// TIA Portal V17 export
// export: Created 2022-07-28T18:02:47.9991032Z, ExportSetting None, DisplayName Totally Integrated Automation Portal, DisplayVersion V17, DisplayName TIA Portal Openness, DisplayVersion V17, DisplayName TIA Portal Teamcenter Gateway, DisplayVersion V17, DisplayName TIA Portal Version Control Interface, DisplayVersion V17, DisplayName TIA Portal Test Suite Advanced, DisplayVersion V17, DisplayName SINAMICS Startdrive Advanced, DisplayVersion V17, DisplayName SINAMICS DCC, DisplayVersion V17, DisplayName SINAMICS Startdrive G130, G150, S120, S150, SINAMICS MV, S210, DisplayVersion V17, DisplayName SINAMICS Startdrive G110M, G120, G120C, G120D, G120P, G115D, DisplayVersion V17, DisplayName STEP 7 Professional, DisplayVersion V17, DisplayName SIMATIC Energy Suite, DisplayVersion V17, DisplayName STEP 7 CFC, DisplayVersion V17, DisplayName STEP 7 Safety, DisplayVersion V17, DisplayName WinCC Advanced / Unified PC, DisplayVersion V17, DisplayName SIMATIC Visualization Architect, DisplayVersion V17
FUNCTION "Field_FC" : Void   // FC19, SCL
{ S7_Optimized_Access := 'TRUE' }
// stored: SetENOAutomatically false
   VAR_TEMP
      t_SupplyRelease : Bool;   // 1 - Release from supply
   END_VAR
BEGIN
   #t_SupplyRelease := true;

   REGION (ID = 1) Витратомір пари на нову рафінацію Steam Flowmeter New
       //Тип елемента: Аналоговий витратомір
       //Параметри давача: Scale=; 4-20mA; Analog = 0 - 27648;
       //Одиниці вимірювання: m3/h
       //Додаткова інформація: SITRANS FX330 / 7ME2610-3LD00-0AA0-Z

       REGION Блок керування       
           "D_SteamFlowmeterNew_FT1_Ctrl"(I_Initialization := "D_General_ProgramDATA".RestartPLC,
                                          IR_Raw := "D_InOut"."SteamFlowmeterNew_FT1".II_AnalogValue,
                                          IR_Coef:=60.0,
                                          II_Mode := 0,
                                          I_GlobalRST := "D_General_ProgramDATA".ResetGlobal,
                                          I_Puls_1s:="D_PLC".PLS.P1S,
                                          IR_CycleTime := "D_PLC".TIME_TCK.cyclic_sec_R,
                                          II_Obj_ID := 1,
                                          IQ_PLC_CycleInfo := "D_PLC_CycleInfo_DATA".Grp_Obj[1, 0]);
       END_REGION

   END_REGION

   REGION (ID = 2) Витратомір пари на стару рафінацію Steam Flowmeter Old
       //Тип елемента: Аналоговий витратомір
       //Параметри давача: Scale=; 4-20mA; Analog = 0 - 27648;
       //Одиниці вимірювання: m3/h
       //Додаткова інформація: SITRANS FX330 / 7ME2610-3LD00-0AA0-Z

       REGION Блок керування       
           "D_SteamFlowmeterOld_FT1_Ctrl"(I_Initialization := "D_General_ProgramDATA".RestartPLC,
                                          IR_Raw := "D_InOut"."SteamFlowmeterOld_FT1".II_AnalogValue,
                                          IR_Coef:=60.0,
                                          II_Mode := 0,
                                          I_GlobalRST := "D_General_ProgramDATA".ResetGlobal,
                                          I_Puls_1s:="D_PLC".PLS.P1S,
                                          IR_CycleTime := "D_PLC".TIME_TCK.cyclic_sec_R,
                                          II_Obj_ID := 2,
                                          IQ_PLC_CycleInfo := "D_PLC_CycleInfo_DATA".Grp_Obj[1, 0]);
       END_REGION

   END_REGION

   REGION (ID = 3) Перетворювач тиску обор.води PTНГр
       //Тип елемента: Аналоговий сигнал
       //Параметри давача: Scale=0-10bar; 4-20mA; Analog = 0 - 27648;
       //Одиниці вимірювання: bar
       //Додаткова інформація: 

       REGION Блок керування       
           "D_PTNGr_PT1_Ctrl"(I_Initialization := "D_General_ProgramDATA".RestartPLC,
                              IR_Raw := "D_InOut"."PTNGr_PT1".II_AnalogValue,
                              II_Mode := 0,
                              I_GlobalRST := "D_General_ProgramDATA".ResetGlobal,
                              IR_CycleTime := "D_PLC".TIME_TCK.cyclic_sec_R,
                              II_Obj_ID := 3,
                              IQ_PLC_CycleInfo := "D_PLC_CycleInfo_DATA".Grp_Obj[1, 0]);
       END_REGION

   END_REGION

   REGION (ID = 4) Перетворювач температури вих.води ХМ1 ТТW1011
       //Тип елемента: Аналоговий сигнал
       //Параметри давача: Scale=0-150C; 4-20mA; Analog = 0 - 27648;
       //Одиниці вимірювання: C
       //Додаткова інформація: 

       REGION Блок керування       
           "D_TTW1011_TT1_Ctrl"(I_Initialization := "D_General_ProgramDATA".RestartPLC,
                                IR_Raw := "D_InOut"."TTW1011_TT1".II_AnalogValue,
                                II_Mode := 0,
                                I_GlobalRST := "D_General_ProgramDATA".ResetGlobal,
                                IR_CycleTime := "D_PLC".TIME_TCK.cyclic_sec_R,
                                II_Obj_ID := 4,
                                IQ_PLC_CycleInfo := "D_PLC_CycleInfo_DATA".Grp_Obj[1, 0]);
       END_REGION

   END_REGION

   REGION (ID = 5) Перетворювач температури вих.води ХМ2 TT811
       //Тип елемента: Аналоговий сигнал
       //Параметри давача: Scale=0-150C; 4-20mA; Analog = 0 - 27648;
       //Одиниці вимірювання: C
       //Додаткова інформація: 

       REGION Блок керування       
           "D_TT811_TT1_Ctrl"(I_Initialization := "D_General_ProgramDATA".RestartPLC,
                              IR_Raw := "D_InOut"."TT811_TT1".II_AnalogValue,
                              II_Mode := 0,
                              I_GlobalRST := "D_General_ProgramDATA".ResetGlobal,
                              IR_CycleTime := "D_PLC".TIME_TCK.cyclic_sec_R,
                              II_Obj_ID := 5,
                              IQ_PLC_CycleInfo := "D_PLC_CycleInfo_DATA".Grp_Obj[1, 0]);
       END_REGION

   END_REGION

   REGION (ID = 6) Перетворювач тиску (рівень басейну градирні 1) LTБ1Гр
       //Тип елемента: Аналоговий сигнал
       //Параметри давача: Scale=0-0.25bar; 4-20mA; Analog = 0 - 27648;
       //Одиниці вимірювання: м
       //Додаткова інформація: 

       REGION Блок керування       
           "D_LTB1Gr_LT1_Ctrl"(I_Initialization := "D_General_ProgramDATA".RestartPLC,
                               IR_Raw := "D_InOut"."LTB1Gr_LT1".II_AnalogValue,
                               II_Mode := 0,
                               I_GlobalRST := "D_General_ProgramDATA".ResetGlobal,
                               IR_CycleTime := "D_PLC".TIME_TCK.cyclic_sec_R,
                               II_Obj_ID := 6,
                               IQ_PLC_CycleInfo := "D_PLC_CycleInfo_DATA".Grp_Obj[1, 0]);
       END_REGION

   END_REGION

   REGION (ID = 7) Перетворювач тиску (рівень басейну градирні 2) LTБ2Гр
       //Тип елемента: Аналоговий сигнал
       //Параметри давача: Scale=0-0.25bar; 4-20mA; Analog = 0 - 27648;
       //Одиниці вимірювання: м
       //Додаткова інформація: 
       //"D_LTB1Gr_LT1_HMI".Config.r_Offset := 1.0;
       REGION Блок керування       
           "D_LTB2Gr_LT1_Ctrl"(I_Initialization := "D_General_ProgramDATA".RestartPLC,
                               IR_Raw := "D_InOut"."LTB2Gr_LT1".II_AnalogValue,
                               II_Mode := 0,
                               I_GlobalRST := "D_General_ProgramDATA".ResetGlobal,
                               IR_CycleTime := "D_PLC".TIME_TCK.cyclic_sec_R,
                               II_Obj_ID := 7,
                               IQ_PLC_CycleInfo := "D_PLC_CycleInfo_DATA".Grp_Obj[1, 0]);
       END_REGION

   END_REGION

   REGION (ID = 8) Аналоговий сигнал від AirForce 1 G1
       //Тип елемента: Аналоговий сигнал
       //Параметри давача: Scale= ; 4-20mA; Analog = 0 - 27648;
       //Одиниці вимірювання: 
       //Додаткова інформація: 

       REGION Блок керування       
           "D_G1_AI1_Ctrl"(I_Initialization := "D_General_ProgramDATA".RestartPLC,
                           IR_Raw := "D_InOut"."G1_AI1".II_AnalogValue,
                           II_Mode := 0,
                           I_GlobalRST := "D_General_ProgramDATA".ResetGlobal,
                           IR_CycleTime := "D_PLC".TIME_TCK.cyclic_sec_R,
                           II_Obj_ID := 8,
                           IQ_PLC_CycleInfo := "D_PLC_CycleInfo_DATA".Grp_Obj[1, 0]);
       END_REGION

   END_REGION

   REGION (ID = 9) Аналоговий сигнал від AirForce 2 G1
       //Тип елемента: Аналоговий сигнал
       //Параметри давача: Scale= ; 4-20mA; Analog = 0 - 27648;
       //Одиниці вимірювання: 
       //Додаткова інформація: 

       REGION Блок керування       
           "D_G1_AI2_Ctrl"(I_Initialization := "D_General_ProgramDATA".RestartPLC,
                           IR_Raw := "D_InOut"."G1_AI2".II_AnalogValue,
                           II_Mode := 0,
                           I_GlobalRST := "D_General_ProgramDATA".ResetGlobal,
                           IR_CycleTime := "D_PLC".TIME_TCK.cyclic_sec_R,
                           II_Obj_ID := 9,
                           IQ_PLC_CycleInfo := "D_PLC_CycleInfo_DATA".Grp_Obj[1, 0]);
       END_REGION

   END_REGION

   REGION (ID = 10) Аналоговий сигнал від AirForce 3 G1
       //Тип елемента: Аналоговий сигнал
       //Параметри давача: Scale= ; 4-20mA; Analog = 0 - 27648;
       //Одиниці вимірювання: 
       //Додаткова інформація: 

       REGION Блок керування       
           "D_G1_AI3_Ctrl"(I_Initialization := "D_General_ProgramDATA".RestartPLC,
                           IR_Raw := "D_InOut"."G1_AI3".II_AnalogValue,
                           II_Mode := 0,
                           I_GlobalRST := "D_General_ProgramDATA".ResetGlobal,
                           IR_CycleTime := "D_PLC".TIME_TCK.cyclic_sec_R,
                           II_Obj_ID := 10,
                           IQ_PLC_CycleInfo := "D_PLC_CycleInfo_DATA".Grp_Obj[1, 0]);
       END_REGION

   END_REGION

   REGION (ID = 11) Аналоговий сигнал від AirForce 4 G1
       //Тип елемента: Аналоговий сигнал
       //Параметри давача: Scale= ; 4-20mA; Analog = 0 - 27648;
       //Одиниці вимірювання: 
       //Додаткова інформація: 

       REGION Блок керування       
           "D_G1_AI4_Ctrl"(I_Initialization := "D_General_ProgramDATA".RestartPLC,
                           IR_Raw := "D_InOut"."G1_AI4".II_AnalogValue,
                           II_Mode := 0,
                           I_GlobalRST := "D_General_ProgramDATA".ResetGlobal,
                           IR_CycleTime := "D_PLC".TIME_TCK.cyclic_sec_R,
                           II_Obj_ID := 11,
                           IQ_PLC_CycleInfo := "D_PLC_CycleInfo_DATA".Grp_Obj[1, 0]);
       END_REGION

   END_REGION

   REGION (ID = 12) Аналоговий сигнал від AirForce 5 G1
       //Тип елемента: Аналоговий сигнал
       //Параметри давача: Scale= ; 4-20mA; Analog = 0 - 27648;
       //Одиниці вимірювання: 
       //Додаткова інформація: 

       REGION Блок керування       
           "D_G1_AI5_Ctrl"(I_Initialization := "D_General_ProgramDATA".RestartPLC,
                           IR_Raw := "D_InOut"."G1_AI5".II_AnalogValue,
                           II_Mode := 0,
                           I_GlobalRST := "D_General_ProgramDATA".ResetGlobal,
                           IR_CycleTime := "D_PLC".TIME_TCK.cyclic_sec_R,
                           II_Obj_ID := 12,
                           IQ_PLC_CycleInfo := "D_PLC_CycleInfo_DATA".Grp_Obj[1, 0]);
       END_REGION

   END_REGION

   REGION (ID = 13) Аналоговий сигнал від AirForce 6 G1
       //Тип елемента: Аналоговий сигнал
       //Параметри давача: Scale= ; 4-20mA; Analog = 0 - 27648;
       //Одиниці вимірювання: 
       //Додаткова інформація: 

       REGION Блок керування       
           "D_G1_AI6_Ctrl"(I_Initialization := "D_General_ProgramDATA".RestartPLC,
                           IR_Raw := "D_InOut"."G1_AI6".II_AnalogValue,
                           II_Mode := 0,
                           I_GlobalRST := "D_General_ProgramDATA".ResetGlobal,
                           IR_CycleTime := "D_PLC".TIME_TCK.cyclic_sec_R,
                           II_Obj_ID := 13,
                           IQ_PLC_CycleInfo := "D_PLC_CycleInfo_DATA".Grp_Obj[1, 0]);
       END_REGION

   END_REGION

   REGION (ID = 14) Перетворювач тиску (рівень ємності конденсату) LT R46
       //Тип елемента: Аналоговий сигнал
       //Параметри давача: Scale=0-0.4bar; 4-20mA; Analog = 0 - 27648;
       //Одиниці вимірювання: м
       //Додаткова інформація: 

       REGION Блок керування       
           "D_LTR46_LT1_Ctrl"(I_Initialization := "D_General_ProgramDATA".RestartPLC,
                              IR_Raw := "D_Filter_LTR46_LT1".qr_Output, //"D_InOut"."LTR46_LT1".II_AnalogValue,
                              II_Mode := 0,
                              I_GlobalRST := "D_General_ProgramDATA".ResetGlobal,
                              IR_CycleTime := "D_PLC".TIME_TCK.cyclic_sec_R,
                              II_Obj_ID := 14,
                              IQ_PLC_CycleInfo := "D_PLC_CycleInfo_DATA".Grp_Obj[1, 0]);
       END_REGION

   END_REGION

   REGION (ID = 15) Температура конденсату TT R46
       //Тип елемента: Аналоговий сигнал
       //Параметри давача: Scale=0-150C; 4-20mA; Analog = 0 - 27648;
       //Одиниці вимірювання: C
       //Додаткова інформація: 

       REGION Блок керування       
           "D_TTR46_TT1_Ctrl"(I_Initialization := "D_General_ProgramDATA".RestartPLC,
                              IR_Raw := "D_InOut"."TTR46_TT1".II_AnalogValue,
                              II_Mode := 0,
                              I_GlobalRST := "D_General_ProgramDATA".ResetGlobal,
                              IR_CycleTime := "D_PLC".TIME_TCK.cyclic_sec_R,
                              II_Obj_ID := 15,
                              IQ_PLC_CycleInfo := "D_PLC_CycleInfo_DATA".Grp_Obj[1, 0]);
       END_REGION

   END_REGION

   REGION (ID = 16) Тиск повітря 1 PT AirLow
       //Тип елемента: Аналоговий сигнал
       //Параметри давача: Scale=0-10bar; 4-20mA; Analog = 0 - 27648;
       //Одиниці вимірювання: bar
       //Додаткова інформація: 

       REGION Блок керування       
           "D_PT_AirLow_PT1_Ctrl"(I_Initialization := "D_General_ProgramDATA".RestartPLC,
                                  IR_Raw := "D_InOut"."PT_AirLow_PT1".II_AnalogValue,
                                  II_Mode := 0,
                                  I_GlobalRST := "D_General_ProgramDATA".ResetGlobal,
                                  IR_CycleTime := "D_PLC".TIME_TCK.cyclic_sec_R,
                                  II_Obj_ID := 16,
                                  IQ_PLC_CycleInfo := "D_PLC_CycleInfo_DATA".Grp_Obj[1, 0]);
       END_REGION

   END_REGION

   REGION (ID = 17) Тиск повітря 2 PT AirHigh
       //Тип елемента: Аналоговий сигнал
       //Параметри давача: Scale=0-10bar; 4-20mA; Analog = 0 - 27648;
       //Одиниці вимірювання: bar
       //Додаткова інформація: 

       REGION Блок керування       
           "D_PT_AirHigh_PT1_Ctrl"(I_Initialization := "D_General_ProgramDATA".RestartPLC,
                                   IR_Raw := "D_InOut"."PT_AirHigh_PT1".II_AnalogValue,
                                   II_Mode := 0,
                                   I_GlobalRST := "D_General_ProgramDATA".ResetGlobal,
                                   IR_CycleTime := "D_PLC".TIME_TCK.cyclic_sec_R,
                                   II_Obj_ID := 17,
                                   IQ_PLC_CycleInfo := "D_PLC_CycleInfo_DATA".Grp_Obj[1, 0]);
       END_REGION

   END_REGION

   REGION (ID = 18) Тиск газу PT Gas
       //Тип елемента: Аналоговий сигнал
       //Параметри давача: Scale= ;4-20ma; Analog = 0 - 27648;
       //Одиниці вимірювання: 
       //Додаткова інформація: 

       REGION Блок керування       
           "D_PT_Gas_PT1_Ctrl"(I_Initialization := "D_General_ProgramDATA".RestartPLC,
                               IR_Raw := "D_InOut"."PT_Gas_PT1".II_AnalogValue,
                               II_Mode := 0,
                               I_GlobalRST := "D_General_ProgramDATA".ResetGlobal,
                               IR_CycleTime := "D_PLC".TIME_TCK.cyclic_sec_R,
                               II_Obj_ID := 18,
                               IQ_PLC_CycleInfo := "D_PLC_CycleInfo_DATA".Grp_Obj[1, 0]);
       END_REGION

   END_REGION

   REGION (ID = 19) Тиск азоту PT Nitrogen
       //Тип елемента: Аналоговий сигнал
       //Параметри давача: Scale= ;4-20ma; Analog = 0 - 27648;
       //Одиниці вимірювання: 
       //Додаткова інформація: 

       REGION Блок керування       
           "D_PT_Nitrogen_PT1_Ctrl"(I_Initialization := "D_General_ProgramDATA".RestartPLC,
                                    IR_Raw := "D_InOut"."PT_Nitrogen_PT1".II_AnalogValue,
                                    II_Mode := 0,
                                    I_GlobalRST := "D_General_ProgramDATA".ResetGlobal,
                                    IR_CycleTime := "D_PLC".TIME_TCK.cyclic_sec_R,
                                    II_Obj_ID := 19,
                                    IQ_PLC_CycleInfo := "D_PLC_CycleInfo_DATA".Grp_Obj[1, 0]);
       END_REGION

   END_REGION

   REGION (ID = 20) Тиск води осмотичної PT W10_1
       //Тип елемента: Аналоговий сигнал
       //Параметри давача: Scale=0-6bar; 4-20mA; Analog = 0 - 27648;
       //Одиниці вимірювання: bar
       //Додаткова інформація: 

       REGION Блок керування       
           "D_PT_W10_1_PT1_Ctrl"(I_Initialization := "D_General_ProgramDATA".RestartPLC,
                                 IR_Raw := "D_InOut"."PT_W10_1_PT1".II_AnalogValue,
                                 II_Mode := 0,
                                 I_GlobalRST := "D_General_ProgramDATA".ResetGlobal,
                                 IR_CycleTime := "D_PLC".TIME_TCK.cyclic_sec_R,
                                 II_Obj_ID := 20,
                                 IQ_PLC_CycleInfo := "D_PLC_CycleInfo_DATA".Grp_Obj[1, 0]);
       END_REGION

   END_REGION

   REGION (ID = 21) Тиск води технічної PT water
       //Тип елемента: Аналоговий сигнал
       //Параметри давача: Scale=0-6bar; 4-20mA; Analog = 0 - 27648;
       //Одиниці вимірювання: bar
       //Додаткова інформація: 

       REGION Блок керування       
           "D_PT_water_PT1_Ctrl"(I_Initialization := "D_General_ProgramDATA".RestartPLC,
                                 IR_Raw := "D_InOut"."PT_water_PT1".II_AnalogValue,
                                 II_Mode := 0,
                                 I_GlobalRST := "D_General_ProgramDATA".ResetGlobal,
                                 IR_CycleTime := "D_PLC".TIME_TCK.cyclic_sec_R,
                                 II_Obj_ID := 21,
                                 IQ_PLC_CycleInfo := "D_PLC_CycleInfo_DATA".Grp_Obj[1, 0]);
       END_REGION

   END_REGION

   REGION (ID = 22) Тиск пари 1 PT steam 1
       //Тип елемента: Аналоговий сигнал
       //Параметри давача: Scale= ;4-20ma; Analog = 0 - 27648;
       //Одиниці вимірювання: 
       //Додаткова інформація: 

       REGION Блок керування       
           "D_PT_steam_1_PT1_Ctrl"(I_Initialization := "D_General_ProgramDATA".RestartPLC,
                                   IR_Raw := "D_InOut"."PT_steam_1_PT1".II_AnalogValue,
                                   II_Mode := 0,
                                   I_GlobalRST := "D_General_ProgramDATA".ResetGlobal,
                                   IR_CycleTime := "D_PLC".TIME_TCK.cyclic_sec_R,
                                   II_Obj_ID := 22,
                                   IQ_PLC_CycleInfo := "D_PLC_CycleInfo_DATA".Grp_Obj[1, 0]);
       END_REGION

   END_REGION

   REGION (ID = 23) Тиск пари 2 PT steam 2
       //Тип елемента: Аналоговий сигнал
       //Параметри давача: Scale= ;4-20ma; Analog = 0 - 27648;
       //Одиниці вимірювання: 
       //Додаткова інформація: 

       REGION Блок керування       
           "D_PT_steam_2_PT1_Ctrl"(I_Initialization := "D_General_ProgramDATA".RestartPLC,
                                   IR_Raw := "D_InOut"."PT_steam_2_PT1".II_AnalogValue,
                                   II_Mode := 0,
                                   I_GlobalRST := "D_General_ProgramDATA".ResetGlobal,
                                   IR_CycleTime := "D_PLC".TIME_TCK.cyclic_sec_R,
                                   II_Obj_ID := 23,
                                   IQ_PLC_CycleInfo := "D_PLC_CycleInfo_DATA".Grp_Obj[1, 0]);
       END_REGION

   END_REGION

   REGION (ID = 24) Тиск пари 3 PT steam 3
       //Тип елемента: Аналоговий сигнал
       //Параметри давача: Scale= ;4-20ma; Analog = 0 - 27648;
       //Одиниці вимірювання: 
       //Додаткова інформація: 

       REGION Блок керування       
           "D_PT_steam_3_PT1_Ctrl"(I_Initialization := "D_General_ProgramDATA".RestartPLC,
                                   IR_Raw := "D_InOut"."PT_steam_3_PT1".II_AnalogValue,
                                   II_Mode := 0,
                                   I_GlobalRST := "D_General_ProgramDATA".ResetGlobal,
                                   IR_CycleTime := "D_PLC".TIME_TCK.cyclic_sec_R,
                                   II_Obj_ID := 24,
                                   IQ_PLC_CycleInfo := "D_PLC_CycleInfo_DATA".Grp_Obj[1, 0]);
       END_REGION

   END_REGION

   REGION (ID = 25) Тиск теплоносія 1 PT coolant 1
       //Тип елемента: Аналоговий сигнал
       //Параметри давача: Scale= ;4-20ma; Analog = 0 - 27648;
       //Одиниці вимірювання: 
       //Додаткова інформація: 

       REGION Блок керування       
           "D_PT_coolant_1_PT1_Ctrl"(I_Initialization := "D_General_ProgramDATA".RestartPLC,
                                     IR_Raw := "D_InOut"."PT_coolant_1_PT1".II_AnalogValue,
                                     II_Mode := 0,
                                     I_GlobalRST := "D_General_ProgramDATA".ResetGlobal,
                                     IR_CycleTime := "D_PLC".TIME_TCK.cyclic_sec_R,
                                     II_Obj_ID := 25,
                                     IQ_PLC_CycleInfo := "D_PLC_CycleInfo_DATA".Grp_Obj[1, 0]);
       END_REGION

   END_REGION

   REGION (ID = 26) Тиск теплоносія 2 PT coolant 2
       //Тип елемента: Аналоговий сигнал
       //Параметри давача: Scale= ;4-20ma; Analog = 0 - 27648;
       //Одиниці вимірювання: 
       //Додаткова інформація: 

       REGION Блок керування       
           "D_PT_coolant_2_PT1_Ctrl"(I_Initialization := "D_General_ProgramDATA".RestartPLC,
                                     IR_Raw := "D_InOut"."PT_coolant_2_PT1".II_AnalogValue,
                                     II_Mode := 0,
                                     I_GlobalRST := "D_General_ProgramDATA".ResetGlobal,
                                     IR_CycleTime := "D_PLC".TIME_TCK.cyclic_sec_R,
                                     II_Obj_ID := 26,
                                     IQ_PLC_CycleInfo := "D_PLC_CycleInfo_DATA".Grp_Obj[1, 0]);
       END_REGION

   END_REGION

   REGION (ID = 27) Температура теплоносія 1 TT coolant 1
       //Тип елемента: Аналоговий сигнал
       //Параметри давача: Scale=0-150C; 4-20mA; Analog = 0 - 27648;
       //Одиниці вимірювання: C
       //Додаткова інформація: 

       REGION Блок керування       
           "D_TT_coolant_1_TT1_Ctrl"(I_Initialization := "D_General_ProgramDATA".RestartPLC,
                                     IR_Raw := "D_InOut"."TT_coolant_1_TT1".II_AnalogValue,
                                     II_Mode := 0,
                                     I_GlobalRST := "D_General_ProgramDATA".ResetGlobal,
                                     IR_CycleTime := "D_PLC".TIME_TCK.cyclic_sec_R,
                                     II_Obj_ID := 27,
                                     IQ_PLC_CycleInfo := "D_PLC_CycleInfo_DATA".Grp_Obj[1, 0]);
       END_REGION

   END_REGION

   REGION (ID = 28) Температура теплоносія 2 TT coolant 2
       //Тип елемента: Аналоговий сигнал
       //Параметри давача: Scale=0-150C; 4-20mA; Analog = 0 - 27648;
       //Одиниці вимірювання: C
       //Додаткова інформація: 

       REGION Блок керування       
           "D_TT_coolant_2_TT1_Ctrl"(I_Initialization := "D_General_ProgramDATA".RestartPLC,
                                     IR_Raw := "D_InOut"."TT_coolant_2_TT1".II_AnalogValue,
                                     II_Mode := 0,
                                     I_GlobalRST := "D_General_ProgramDATA".ResetGlobal,
                                     IR_CycleTime := "D_PLC".TIME_TCK.cyclic_sec_R,
                                     II_Obj_ID := 28,
                                     IQ_PLC_CycleInfo := "D_PLC_CycleInfo_DATA".Grp_Obj[1, 0]);
       END_REGION

   END_REGION

   REGION (ID = 29) Перетворювач тиску подачі  кислоти PT PW579CA
       //Тип елемента: Аналоговий сигнал
       //Параметри давача: Scale=0-6bar; 4-20mA; Analog = 0 - 27648;
       //Одиниці вимірювання: bar
       //Додаткова інформація: 

       REGION Блок керування       
           "D_PT_PW579CA_PT1_Ctrl"(I_Initialization := "D_General_ProgramDATA".RestartPLC,
                                   IR_Raw := "D_InOut"."PT_PW579CA_PT1".II_AnalogValue,
                                   II_Mode := 0,
                                   I_GlobalRST := "D_General_ProgramDATA".ResetGlobal,
                                   IR_CycleTime := "D_PLC".TIME_TCK.cyclic_sec_R,
                                   II_Obj_ID := 29,
                                   IQ_PLC_CycleInfo := "D_PLC_CycleInfo_DATA".Grp_Obj[1, 0]);
       END_REGION

   END_REGION

   REGION (ID = 30) Рівень в ємності лимонної кислоти LT PW579CA
       //Тип елемента: Аналоговий сигнал
       //Параметри давача: Scale=0-0.1bar; 4-20mA; Analog = 0 - 27648;
       //Одиниці вимірювання: м
       //Додаткова інформація: 

       REGION Блок керування       
           "D_LT_PW579CA_LT1_Ctrl"(I_Initialization := "D_General_ProgramDATA".RestartPLC,
                                   IR_Raw := "D_InOut"."LT_PW579CA_LT1".II_AnalogValue,
                                   II_Mode := 0,
                                   I_GlobalRST := "D_General_ProgramDATA".ResetGlobal,
                                   IR_CycleTime := "D_PLC".TIME_TCK.cyclic_sec_R,
                                   II_Obj_ID := 30,
                                   IQ_PLC_CycleInfo := "D_PLC_CycleInfo_DATA".Grp_Obj[1, 0]);
       END_REGION

   END_REGION

   REGION (ID = 31) Перетворювач тиску подачі  лугу PT PW579NA
       //Тип елемента: Аналоговий сигнал
       //Параметри давача: Scale=0-6bar; 4-20mA; Analog = 0 - 27648;
       //Одиниці вимірювання: bar
       //Додаткова інформація: 

       REGION Блок керування       
           "D_PT_PW579NA_PT1_Ctrl"(I_Initialization := "D_General_ProgramDATA".RestartPLC,
                                   IR_Raw := "D_InOut"."PT_PW579NA_PT1".II_AnalogValue,
                                   II_Mode := 0,
                                   I_GlobalRST := "D_General_ProgramDATA".ResetGlobal,
                                   IR_CycleTime := "D_PLC".TIME_TCK.cyclic_sec_R,
                                   II_Obj_ID := 31,
                                   IQ_PLC_CycleInfo := "D_PLC_CycleInfo_DATA".Grp_Obj[1, 0]);
       END_REGION

   END_REGION

   REGION (ID = 32) Перетворювач тиску (рівень води в ємності) LT W10 OW
       //Тип елемента: Аналоговий сигнал
       //Параметри давача: Scale=0-0.25bar; 4-20mA; Analog = 0 - 27648;
       //Одиниці вимірювання: м
       //Додаткова інформація: 

       REGION Блок керування       
           "D_LT_W10_OW_LT1_Ctrl"(I_Initialization := "D_General_ProgramDATA".RestartPLC,
                                  IR_Raw := "D_InOut"."LT_W10_OW_LT1".II_AnalogValue,
                                   IR_High:=27648, //17280.0
                                  II_Mode := 0,
                                  I_GlobalRST := "D_General_ProgramDATA".ResetGlobal,
                                  IR_CycleTime := "D_PLC".TIME_TCK.cyclic_sec_R,
                                  II_Obj_ID := 32,
                                  IQ_PLC_CycleInfo := "D_PLC_CycleInfo_DATA".Grp_Obj[1, 0]);
       END_REGION

   END_REGION

   REGION (ID = 33) Температура води охолодження дублюючого насоса TT P822 2
       //Тип елемента: Аналоговий сигнал
       //Параметри давача: Scale= ; 4-20mA; Analog = 0 - 27648;
       //Одиниці вимірювання: C
       //Додаткова інформація: 

       REGION Блок керування       
           "D_TT_P822_2_TT1_Ctrl"(I_Initialization := "D_General_ProgramDATA".RestartPLC,
                                  IR_Raw := "D_InOut"."TT_P822_2_TT1".II_AnalogValue,
                                  II_Mode := 0,
                                  I_GlobalRST := "D_General_ProgramDATA".ResetGlobal,
                                  IR_CycleTime := "D_PLC".TIME_TCK.cyclic_sec_R,
                                  II_Obj_ID := 33,
                                  IQ_PLC_CycleInfo := "D_PLC_CycleInfo_DATA".Grp_Obj[1, 0]);
       END_REGION

   END_REGION

   REGION (ID = 36) Дискретний сигнал від AirForce 1 G1
       //Тип елемента: Дискретний сигнал
       //Параметри давача: Info;NO;
       //Додаткова інформація: 

       REGION Блок керування
           "D_G1_DI1_Ctrl"(I_Initialization := "D_General_ProgramDATA".RestartPLC,
                           I_Raw := "D_InOut"."G1_DI1".DescreteValue,
                           II_Mode := 4,
                           I_GlobalRST := "D_General_ProgramDATA".ResetGlobal,
                           IR_CycleTime := "D_PLC".TIME_TCK.cyclic_sec_R,
                           II_Obj_ID := 36,
                           IO_PLC_CycleInfo := "D_PLC_CycleInfo_DATA".Grp_Obj[1, 0]);
       END_REGION

   END_REGION

   REGION (ID = 37) Дискретний сигнал від AirForce 2 G1
       //Тип елемента: Дискретний сигнал
       //Параметри давача: Info;NO;
       //Додаткова інформація: 

       REGION Блок керування
           "D_G1_DI2_Ctrl"(I_Initialization := "D_General_ProgramDATA".RestartPLC,
                           I_Raw := "D_InOut"."G1_DI2".DescreteValue,
                           II_Mode := 4,
                           I_GlobalRST := "D_General_ProgramDATA".ResetGlobal,
                           IR_CycleTime := "D_PLC".TIME_TCK.cyclic_sec_R,
                           II_Obj_ID := 37,
                           IO_PLC_CycleInfo := "D_PLC_CycleInfo_DATA".Grp_Obj[1, 0]);
       END_REGION

   END_REGION

   REGION (ID = 38) Дискретний сигнал від AirForce 3 G1
       //Тип елемента: Дискретний сигнал
       //Параметри давача: Info;NO;
       //Додаткова інформація: 

       REGION Блок керування
           "D_G1_DI3_Ctrl"(I_Initialization := "D_General_ProgramDATA".RestartPLC,
                           I_Raw := "D_InOut"."G1_DI3".DescreteValue,
                           II_Mode := 4,
                           I_GlobalRST := "D_General_ProgramDATA".ResetGlobal,
                           IR_CycleTime := "D_PLC".TIME_TCK.cyclic_sec_R,
                           II_Obj_ID := 38,
                           IO_PLC_CycleInfo := "D_PLC_CycleInfo_DATA".Grp_Obj[1, 0]);
       END_REGION

   END_REGION

   REGION (ID = 39) Дискретний сигнал від AirForce 4 G1
       //Тип елемента: Дискретний сигнал
       //Параметри давача: Info;NO;
       //Додаткова інформація: 

       REGION Блок керування
           "D_G1_DI4_Ctrl"(I_Initialization := "D_General_ProgramDATA".RestartPLC,
                           I_Raw := "D_InOut"."G1_DI4".DescreteValue,
                           II_Mode := 4,
                           I_GlobalRST := "D_General_ProgramDATA".ResetGlobal,
                           IR_CycleTime := "D_PLC".TIME_TCK.cyclic_sec_R,
                           II_Obj_ID := 39,
                           IO_PLC_CycleInfo := "D_PLC_CycleInfo_DATA".Grp_Obj[1, 0]);
       END_REGION

   END_REGION

   REGION (ID = 40) Дискретний сигнал від AirForce 5 G1
       //Тип елемента: Дискретний сигнал
       //Параметри давача: Info;NO;
       //Додаткова інформація: 

       REGION Блок керування
           "D_G1_DI5_Ctrl"(I_Initialization := "D_General_ProgramDATA".RestartPLC,
                           I_Raw := "D_InOut"."G1_DI5".DescreteValue,
                           II_Mode := 4,
                           I_GlobalRST := "D_General_ProgramDATA".ResetGlobal,
                           IR_CycleTime := "D_PLC".TIME_TCK.cyclic_sec_R,
                           II_Obj_ID := 40,
                           IO_PLC_CycleInfo := "D_PLC_CycleInfo_DATA".Grp_Obj[1, 0]);
       END_REGION

   END_REGION

   REGION (ID = 41) Контроль роботи холодильної машини 1 - робота W1011
       //Тип елемента: Дискретний сигнал
       //Параметри давача: Info;NO;
       //Додаткова інформація: 

       REGION Блок керування
           "D_W1011_S1_Ctrl"(I_Initialization := "D_General_ProgramDATA".RestartPLC,
                             //I_Raw := "D_InOut"."W1011_S1".DescreteValue,
                             //II_Mode := 4,
                             I_GlobalRST := "D_General_ProgramDATA".ResetGlobal,
                             IR_CycleTime := "D_PLC".TIME_TCK.cyclic_sec_R,
                             II_Obj_ID := 41,
                             IO_PLC_CycleInfo := "D_PLC_CycleInfo_DATA".Grp_Obj[1, 0]);
       END_REGION

   END_REGION

   REGION (ID = 42) Контроль роботи холодильної машини 1 - аварія W1011
       //Тип елемента: Дискретний сигнал
       //Параметри давача: Err;NO;
       //Додаткова інформація: 

       REGION Блок керування
           "D_W1011_S2_Ctrl"(I_Initialization := "D_General_ProgramDATA".RestartPLC,
                             I_Raw := "D_InOut"."W1011_S2".DescreteValue,
                             II_Mode := 0,
                             I_GlobalRST := "D_General_ProgramDATA".ResetGlobal,
                             IR_CycleTime := "D_PLC".TIME_TCK.cyclic_sec_R,
                             II_Obj_ID := 42,
                             IO_PLC_CycleInfo := "D_PLC_CycleInfo_DATA".Grp_Obj[1, 0]);
       END_REGION

   END_REGION

   REGION (ID = 43) Контроль роботи холодильної машини 2 - робота 811
       //Тип елемента: Дискретний сигнал
       //Параметри давача: Info;NO;
       //Додаткова інформація: 

       REGION Блок керування
           "D_811_S1_Ctrl"(I_Initialization := "D_General_ProgramDATA".RestartPLC,
                           I_Raw := "D_InOut"."811_S1".DescreteValue,
                           II_Mode := 4,
                           I_GlobalRST := "D_General_ProgramDATA".ResetGlobal,
                           IR_CycleTime := "D_PLC".TIME_TCK.cyclic_sec_R,
                           II_Obj_ID := 43,
                           IO_PLC_CycleInfo := "D_PLC_CycleInfo_DATA".Grp_Obj[1, 0]);
       END_REGION

   END_REGION

   REGION (ID = 44) Контроль роботи холодильної машини 2 - аварія 811
       //Тип елемента: Дискретний сигнал
       //Параметри давача: Err;NO;
       //Додаткова інформація: 

       REGION Блок керування
           "D_811_S2_Ctrl"(I_Initialization := "D_General_ProgramDATA".RestartPLC,
                           I_Raw := "D_InOut"."811_S2".DescreteValue,
                           II_Mode := 0,
                           I_GlobalRST := "D_General_ProgramDATA".ResetGlobal,
                           IR_CycleTime := "D_PLC".TIME_TCK.cyclic_sec_R,
                           II_Obj_ID := 44,
                           IO_PLC_CycleInfo := "D_PLC_CycleInfo_DATA".Grp_Obj[1, 0]);
       END_REGION

   END_REGION

   REGION (ID = 45) Парогенератор і бойлерна - загазованість H DI7
       //Тип елемента: Дискретний сигнал
       //Параметри давача: Err;NC;
       //Додаткова інформація: 

       "D_DI7_S1_HMI".Config.WarnDetectTime := 0.0;
       "D_DI7_S1_HMI".Config.AutoReset := true;
       REGION Блок керування
           "D_DI7_S1_Ctrl"(I_Initialization := "D_General_ProgramDATA".RestartPLC,
                           I_Raw := "D_InOut"."DI7_S1".DescreteValue,
                           II_Mode := 1,
                           I_GlobalRST := "D_General_ProgramDATA".ResetGlobal,
                           IR_CycleTime := "D_PLC".TIME_TCK.cyclic_sec_R,
                           II_Obj_ID := 45,
                           IO_PLC_CycleInfo := "D_PLC_CycleInfo_DATA".Grp_Obj[1, 0]);
       END_REGION

   END_REGION

   REGION (ID = 46) Парогенератор і бойлерна - аварія DI7
       //Тип елемента: Дискретний сигнал
       //Параметри давача: Err;NC;
       //Додаткова інформація: 

       REGION Блок керування
           "D_DI7_S2_Ctrl"(I_Initialization := "D_General_ProgramDATA".RestartPLC,
                           I_Raw := "D_InOut"."DI7_S2".DescreteValue,
                           II_Mode := 1,
                           I_GlobalRST := "D_General_ProgramDATA".ResetGlobal,
                           IR_CycleTime := "D_PLC".TIME_TCK.cyclic_sec_R,
                           II_Obj_ID := 46,
                           IO_PLC_CycleInfo := "D_PLC_CycleInfo_DATA".Grp_Obj[1, 0]);
       END_REGION

   END_REGION

   REGION (ID = 47) Парогенератор і бойлерна - загазованість HH DI7
       //Тип елемента: Дискретний сигнал
       //Параметри давача: Err;NC;
       //Додаткова інформація: 

       "D_DI7_S3_HMI".Config.WarnDetectTime := 0.0;
       "D_DI7_S3_HMI".Config.AutoReset := true;
       REGION Блок керування
           "D_DI7_S3_Ctrl"(I_Initialization := "D_General_ProgramDATA".RestartPLC,
                           I_Raw := "D_InOut"."DI7_S3".DescreteValue,
                           II_Mode := 1,
                           I_GlobalRST := "D_General_ProgramDATA".ResetGlobal,
                           IR_CycleTime := "D_PLC".TIME_TCK.cyclic_sec_R,
                           II_Obj_ID := 47,
                           IO_PLC_CycleInfo := "D_PLC_CycleInfo_DATA".Grp_Obj[1, 0]);
       END_REGION

   END_REGION

   REGION (ID = 48) Протік  води охолодження дублюючого насоса FT P822 2
       //Тип елемента: Дискретний сигнал
       //Параметри давача: Info;NC;
       //Додаткова інформація: 

       REGION Блок керування
           "D_FT_P822_2_FT1_Ctrl"(I_Initialization := "D_General_ProgramDATA".RestartPLC,
                                  I_Raw := "D_InOut"."FT_P822_2_FT1".DescreteValue,
                                  II_Mode := 5,
                                  I_GlobalRST := "D_General_ProgramDATA".ResetGlobal,
                                  IR_CycleTime := "D_PLC".TIME_TCK.cyclic_sec_R,
                                  II_Obj_ID := 48,
                                  IO_PLC_CycleInfo := "D_PLC_CycleInfo_DATA".Grp_Obj[1, 0]);
       END_REGION

   END_REGION
END_FUNCTION
